// TIA Portal project "FactoryIO_Template_S7-1500_V14" (V14)

(* hardware
DEVICE "S71500/ET200MP-Station_1"  S7-1500 station
   slot 0: "Profilschiene_0"  6ES7 590-1***0-0AA0
   slot 1: "PLC_1"  CPU 1511-1 PN  6ES7 511-1AK00-0AB0  V1.8
   slot 2: "AI 8xU/I/RTD/TC ST_1"  AI 8xU/I/RTD/TC ST  6ES7 531-7KF00-0AB0  V2.0
   slot 3: "AI 8xU/I/RTD/TC ST_2"  AI 8xU/I/RTD/TC ST  6ES7 531-7KF00-0AB0  V2.0
   slot 4: "AI 8xU/I/RTD/TC ST_3"  AI 8xU/I/RTD/TC ST  6ES7 531-7KF00-0AB0  V2.0
   slot 5: "AI 8xU/I/RTD/TC ST_4"  AI 8xU/I/RTD/TC ST  6ES7 531-7KF00-0AB0  V2.0
   slot 6: "DI 16x24VDC BA_1"  DI 16x24VDC BA  6ES7 521-1BH10-0AA0  V1.0
*)

// ===== PLC "PLC_1"  CPU 1511-1 PN =====

VAR_GLOBAL   // PLC tag table "Standard-Variablentabelle"
   "start button" AT %I0.0 : Bool;
   "konveyöl 1" AT %Q0.0 : Bool;
   "start ışık" AT %Q0.1 : Bool;
   "Stop button" AT %I0.1 : Bool;
   "stop ışık" AT %Q0.2 : Bool;
   "mavi metaryel sensor" AT %I0.2 : Bool;
   "konveyör mavi yol" AT %Q0.3 : Bool;
   "mavi kemer" AT %Q0.4 : Bool;
   "mavi kol" AT %Q0.5 : Bool;
   "mavi bekleme" AT %Q0.6 : Bool;
   "mavi bekleme sensör baş" AT %I0.3 : Bool;
   "mavie bekleme sensör son" AT %I0.4 : Bool;
   "mavi x hareket" AT %Q0.7 : Bool;
   "mavi hareket z" AT %Q1.0 : Bool;
   "mavi tutucu(1)" AT %Q1.1 : Bool;
   "restart" AT %I0.5 : Bool;
   "depo mavi" AT %Q1.2 : Bool;
   "depo mavi sensor" AT %I0.6 : Bool;
   "mavi depo lamba" AT %Q1.3 : Bool;
   "mavi restart" AT %I0.7 : Bool;
   "konveyör 2" AT %Q1.4 : Bool;
   "konveyör yeşil yol" AT %Q1.5 : Bool;
   "yeşil metaryel sensör" AT %I1.0 : Bool;
   "yeşil kol" AT %Q1.6 : Bool;
   "yeşil kemer" AT %Q1.7 : Bool;
   "yeşil bekleme sensör baş" AT %I1.1 : Bool;
   "yeşil bekleme sensör son" AT %I1.2 : Bool;
   "yeşil bekleme" AT %Q2.0 : Bool;
   "depo mavi sensör" AT %I1.3 : Bool;
   "yeşil x hareket" AT %Q2.1 : Bool;
   "yeşil hareket z" AT %Q2.2 : Bool;
   "yeşil tutucu(1)" AT %Q2.3 : Bool;
   "depo yeşil sensor" AT %I1.4 : Bool;
   "yeşil restart" AT %I1.5 : Bool;
   "depo yeşil" AT %Q2.4 : Bool;
   "depo yeşil lamba" AT %Q2.5 : Bool;
   "Tag_1" AT %M110.0 : Bool;
   "Tag_2" AT %M120.0 : Bool;
   "konveyör metal yol" AT %Q2.6 : Bool;
   "metal metaryel sensör" AT %I1.6 : Bool;
   "metal kol" AT %Q2.7 : Bool;
   "metal kemer" AT %Q3.0 : Bool;
   "metal bekleme baş" AT %I1.7 : Bool;
   "metal bekleme son" AT %I2.0 : Bool;
   "metal bekleme" AT %Q3.1 : Bool;
   "depo metal sensör" AT %I2.1 : Bool;
   "depo metal" AT %Q3.5 : Bool;
   "depo metal lamba" AT %Q3.6 : Bool;
   "Tag_3" AT %M130.0 : Bool;
   "metal restart" AT %I2.2 : Bool;
   "Tag_4" AT %MD140 : Real;
   "Tag_5" AT %QW30 : Word;
   "metal y" AT %QD30 : Real;
   "Tag_7" AT %MD150 : Real;
   "metal z" AT %QD34 : Real;
   "metal tutma" AT %Q3.2 : Bool;
   "Tag_9" AT %MD160 : Real;
   "metal x" AT %QD38 : Real;
END_VAR

// folder: System blocks/Program resources

DATA_BLOCK "mavi"   // DB1
{ S7_Optimized_Access := 'TRUE' }
AUTHOR : Simatic
FAMILY : IEC
NAME : IEC_TMR
VERSION : 1.0
// stored: InstanceOfName IEC_TIMER
"IEC_TIMER"
BEGIN
END_DATA_BLOCK

DATA_BLOCK "mavi depolama"   // DB2
{ S7_Optimized_Access := 'TRUE' }
AUTHOR : Simatic
FAMILY : IEC
NAME : IEC_TMR
VERSION : 1.0
// stored: InstanceOfName IEC_TIMER
"IEC_TIMER"
BEGIN
END_DATA_BLOCK

DATA_BLOCK "mavi tutucu"   // DB3
{ S7_Optimized_Access := 'TRUE' }
AUTHOR : Simatic
FAMILY : IEC
NAME : IEC_TMR
VERSION : 1.0
// stored: InstanceOfName IEC_TIMER
"IEC_TIMER"
BEGIN
END_DATA_BLOCK

DATA_BLOCK "mavi 2"   // DB4
{ S7_Optimized_Access := 'TRUE' }
AUTHOR : Simatic
FAMILY : IEC
NAME : IEC_TMR
VERSION : 1.0
// stored: InstanceOfName IEC_TIMER
"IEC_TIMER"
BEGIN
END_DATA_BLOCK

DATA_BLOCK "mavi 3"   // DB5
{ S7_Optimized_Access := 'TRUE' }
AUTHOR : Simatic
FAMILY : IEC
NAME : IEC_TMR
VERSION : 1.0
// stored: InstanceOfName IEC_TIMER
"IEC_TIMER"
BEGIN
END_DATA_BLOCK

DATA_BLOCK "mavi 4"   // DB6
{ S7_Optimized_Access := 'TRUE' }
AUTHOR : Simatic
FAMILY : IEC
NAME : IEC_TMR
VERSION : 1.0
// stored: InstanceOfName IEC_TIMER
"IEC_TIMER"
BEGIN
END_DATA_BLOCK

DATA_BLOCK "mavi bekleme son sayıcı"   // DB7
{ S7_Optimized_Access := 'TRUE' }
AUTHOR : Simatic
FAMILY : IEC
NAME : CNTR
VERSION : 1.0
// stored: InstanceOfName IEC_COUNTER
"IEC_COUNTER"
BEGIN
END_DATA_BLOCK

DATA_BLOCK "yeşil"   // DB8
{ S7_Optimized_Access := 'TRUE' }
AUTHOR : Simatic
FAMILY : IEC
NAME : IEC_TMR
VERSION : 1.0
// stored: InstanceOfName IEC_TIMER
"IEC_TIMER"
BEGIN
END_DATA_BLOCK

DATA_BLOCK "yeşil depolama"   // DB9
{ S7_Optimized_Access := 'TRUE' }
AUTHOR : Simatic
FAMILY : IEC
NAME : IEC_TMR
VERSION : 1.0
// stored: InstanceOfName IEC_TIMER
"IEC_TIMER"
BEGIN
END_DATA_BLOCK

DATA_BLOCK "yeşil tutucu"   // DB10
{ S7_Optimized_Access := 'TRUE' }
AUTHOR : Simatic
FAMILY : IEC
NAME : IEC_TMR
VERSION : 1.0
// stored: InstanceOfName IEC_TIMER
"IEC_TIMER"
BEGIN
END_DATA_BLOCK

DATA_BLOCK "yeşil 2"   // DB11
{ S7_Optimized_Access := 'TRUE' }
AUTHOR : Simatic
FAMILY : IEC
NAME : IEC_TMR
VERSION : 1.0
// stored: InstanceOfName IEC_TIMER
"IEC_TIMER"
BEGIN
END_DATA_BLOCK

DATA_BLOCK "yeşil 3"   // DB12
{ S7_Optimized_Access := 'TRUE' }
AUTHOR : Simatic
FAMILY : IEC
NAME : IEC_TMR
VERSION : 1.0
// stored: InstanceOfName IEC_TIMER
"IEC_TIMER"
BEGIN
END_DATA_BLOCK

DATA_BLOCK "yeşil 4"   // DB13
{ S7_Optimized_Access := 'TRUE' }
AUTHOR : Simatic
FAMILY : IEC
NAME : IEC_TMR
VERSION : 1.0
// stored: InstanceOfName IEC_TIMER
"IEC_TIMER"
BEGIN
END_DATA_BLOCK

DATA_BLOCK "yeşil bekleme son sayıcı"   // DB14
{ S7_Optimized_Access := 'TRUE' }
AUTHOR : Simatic
FAMILY : IEC
NAME : CNTR
VERSION : 1.0
// stored: InstanceOfName IEC_COUNTER
"IEC_COUNTER"
BEGIN
END_DATA_BLOCK

DATA_BLOCK "mavi sayma"   // DB15
{ S7_Optimized_Access := 'TRUE' }
AUTHOR : Simatic
FAMILY : IEC
NAME : IEC_TMR
VERSION : 1.0
// stored: InstanceOfName IEC_TIMER
"IEC_TIMER"
BEGIN
END_DATA_BLOCK

DATA_BLOCK "yeşil sayma"   // DB16
{ S7_Optimized_Access := 'TRUE' }
AUTHOR : Simatic
FAMILY : IEC
NAME : IEC_TMR
VERSION : 1.0
// stored: InstanceOfName IEC_TIMER
"IEC_TIMER"
BEGIN
END_DATA_BLOCK

DATA_BLOCK "metal"   // DB17
{ S7_Optimized_Access := 'TRUE' }
AUTHOR : Simatic
FAMILY : IEC
NAME : IEC_TMR
VERSION : 1.0
// stored: InstanceOfName IEC_TIMER
"IEC_TIMER"
BEGIN
END_DATA_BLOCK

DATA_BLOCK "metal 1"   // DB18
{ S7_Optimized_Access := 'TRUE' }
AUTHOR : Simatic
FAMILY : IEC
NAME : IEC_TMR
VERSION : 1.0
// stored: InstanceOfName IEC_TIMER
"IEC_TIMER"
BEGIN
END_DATA_BLOCK

DATA_BLOCK "metal 2"   // DB19
{ S7_Optimized_Access := 'TRUE' }
AUTHOR : Simatic
FAMILY : IEC
NAME : IEC_TMR
VERSION : 1.0
// stored: InstanceOfName IEC_TIMER
"IEC_TIMER"
BEGIN
END_DATA_BLOCK

DATA_BLOCK "metal 3"   // DB20
{ S7_Optimized_Access := 'TRUE' }
AUTHOR : Simatic
FAMILY : IEC
NAME : IEC_TMR
VERSION : 1.0
// stored: InstanceOfName IEC_TIMER
"IEC_TIMER"
BEGIN
END_DATA_BLOCK

DATA_BLOCK "metal 4"   // DB21
{ S7_Optimized_Access := 'TRUE' }
AUTHOR : Simatic
FAMILY : IEC
NAME : IEC_TMR
VERSION : 1.0
// stored: InstanceOfName IEC_TIMER
"IEC_TIMER"
BEGIN
END_DATA_BLOCK

DATA_BLOCK "metal 5"   // DB22
{ S7_Optimized_Access := 'TRUE' }
AUTHOR : Simatic
FAMILY : IEC
NAME : IEC_TMR
VERSION : 1.0
// stored: InstanceOfName IEC_TIMER
"IEC_TIMER"
BEGIN
END_DATA_BLOCK

DATA_BLOCK "metal bekleme son sayıcı"   // DB23
{ S7_Optimized_Access := 'TRUE' }
AUTHOR : Simatic
FAMILY : IEC
NAME : CNTR
VERSION : 1.0
// stored: InstanceOfName IEC_COUNTER
"IEC_COUNTER"
BEGIN
END_DATA_BLOCK

DATA_BLOCK "metal sayma"   // DB24
{ S7_Optimized_Access := 'TRUE' }
AUTHOR : Simatic
FAMILY : IEC
NAME : IEC_TMR
VERSION : 1.0
// stored: InstanceOfName IEC_TIMER
"IEC_TIMER"
BEGIN
END_DATA_BLOCK

// folder: (top level)

FUNCTION "MHJ-PLC-Lab-Function-S71500" : Void   // FC9000, SCL
{ S7_Optimized_Access := 'TRUE' }
VERSION : 0.1
   VAR_TEMP
      Value : Byte;
      ForCounter : Int;
   END_VAR
   VAR CONSTANT
      Value_01_DW : DWord := 16#1223_5486;
      Value_02_DW : DWord := 16#A6C9_D1F5;
   END_VAR
BEGIN

   #Value:=PEEK(area := 16#82,
        dbNumber := 0,
        byteOffset := 511);
   #Value := #Value + 1;

   POKE(area := 16#82,
        dbNumber := 0,
        byteOffset := 511,
        value := #Value);

   POKE(area := 16#82,
        dbNumber := 0,
        byteOffset := 1016,
        value := #Value_01_DW);
   POKE(area := 16#82,
        dbNumber := 0,
        byteOffset := 1020,
        value := #Value_02_DW);

   FOR #ForCounter := 0 TO 63 DO
       #Value:=PEEK(area := 16#1,
            dbNumber := 0,
            byteOffset := #ForCounter);
       POKE(area := 16#81,
            dbNumber := 0,
            byteOffset := #ForCounter,
            value := #Value);
   END_FOR;
   #Value := PEEK(area := 16#1,
                  dbNumber := 0,
                  byteOffset := 512);
   POKE(area := 16#82,
        dbNumber := 0,
        byteOffset := 512,
        value := #Value);
END_FUNCTION

ORGANIZATION_BLOCK "Main"   // OB1, LAD, ProgramCycle
TITLE = "Main Program Sweep (Cycle)"
{ S7_Optimized_Access := 'TRUE' }
VERSION : 0.1
   VAR_INPUT
      Initial_Call : Bool;   // Initial call of this OB
      Remanence : Bool;   // =True, if remanent data are available
   END_VAR
   VAR_TEMP   // added for the SCL form of the ladder/FBD networks
      _w1 : Bool;
      _w2 : Bool;
   END_VAR
BEGIN

REGION Network 1
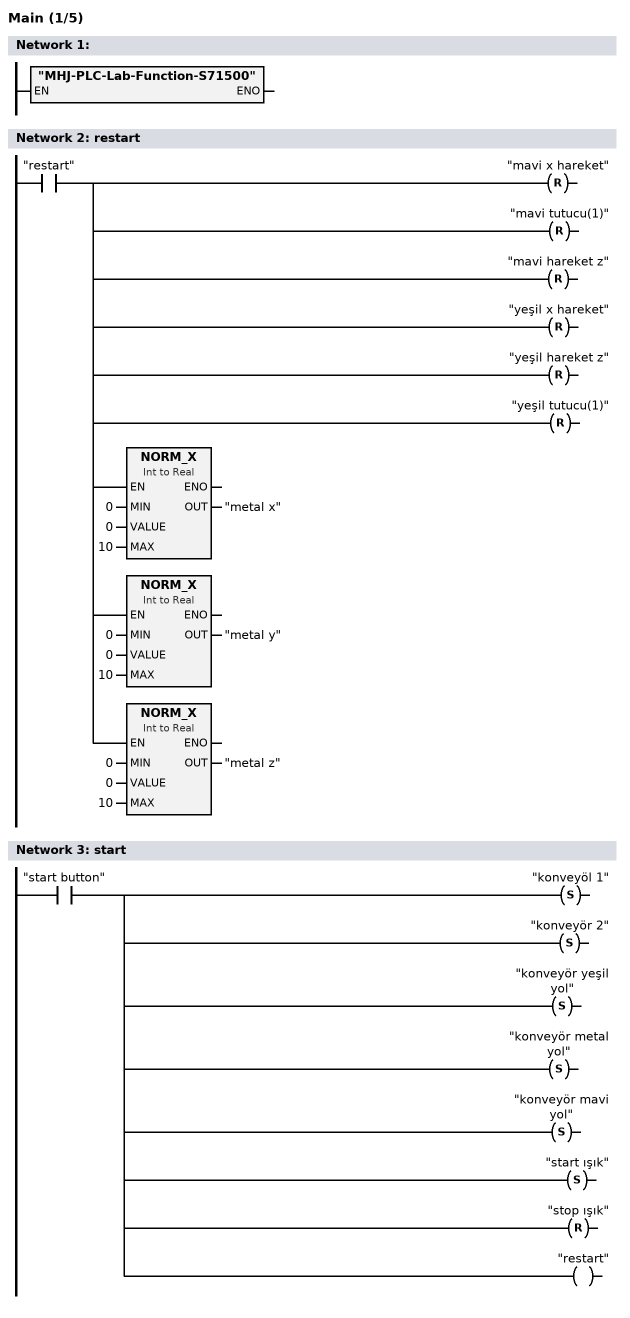
   RUNG wire#powerrail
      "MHJ-PLC-Lab-Function-S71500"()
   END_RUNG
   // the same network as SCL:
   "MHJ-PLC-Lab-Function-S71500"();
END_REGION

REGION Network 2: restart
   RUNG wire#powerrail
      Contact( "restart" )
      wire#w1
      R_Coil( "mavi x hareket" )
   END_RUNG
   RUNG wire#w1
      R_Coil( "mavi tutucu(1)" )
   END_RUNG
   RUNG wire#w1
      R_Coil( "mavi hareket z" )
   END_RUNG
   RUNG wire#w1
      R_Coil( "yeşil x hareket" )
   END_RUNG
   RUNG wire#w1
      R_Coil( "yeşil hareket z" )
   END_RUNG
   RUNG wire#w1
      R_Coil( "yeşil tutucu(1)" )
   END_RUNG
   RUNG wire#w1
      { S7_Templates := "[SrcType := Int, DestType := Real]" } Normalize(min := 0, value := 0, max := 10, out => "metal x")
   END_RUNG
   RUNG wire#w1
      { S7_Templates := "[SrcType := Int, DestType := Real]" } Normalize(min := 0, value := 0, max := 10, out => "metal y")
   END_RUNG
   RUNG wire#w1
      { S7_Templates := "[SrcType := Int, DestType := Real]" } Normalize(min := 0, value := 0, max := 10, out => "metal z")
   END_RUNG
   // the same network as SCL:
   IF "restart" THEN
       "mavi x hareket" := FALSE;
       "mavi tutucu(1)" := FALSE;
       "mavi hareket z" := FALSE;
       "yeşil x hareket" := FALSE;
       "yeşil hareket z" := FALSE;
       "yeşil tutucu(1)" := FALSE;
       "metal x" := NORM_X(MIN := 0, VALUE := 0, MAX := 10);
       "metal y" := NORM_X(MIN := 0, VALUE := 0, MAX := 10);
       "metal z" := NORM_X(MIN := 0, VALUE := 0, MAX := 10);
   END_IF;
END_REGION

REGION Network 3: start
   RUNG wire#powerrail
      Contact( "start button" )
      wire#w1
      S_Coil( "konveyöl 1" )
   END_RUNG
   RUNG wire#w1
      S_Coil( "konveyör 2" )
   END_RUNG
   RUNG wire#w1
      S_Coil( "konveyör yeşil yol" )
   END_RUNG
   RUNG wire#w1
      S_Coil( "konveyör metal yol" )
   END_RUNG
   RUNG wire#w1
      S_Coil( "konveyör mavi yol" )
   END_RUNG
   RUNG wire#w1
      S_Coil( "start ışık" )
   END_RUNG
   RUNG wire#w1
      R_Coil( "stop ışık" )
   END_RUNG
   RUNG wire#w1
      Coil( "restart" )
   END_RUNG
   // the same network as SCL:
   IF "start button" THEN
       "konveyöl 1" := TRUE;
       "konveyör 2" := TRUE;
       "konveyör yeşil yol" := TRUE;
       "konveyör metal yol" := TRUE;
       "konveyör mavi yol" := TRUE;
       "start ışık" := TRUE;
       "stop ışık" := FALSE;
   END_IF;
   "restart" := "start button";
END_REGION

REGION Network 4: stop
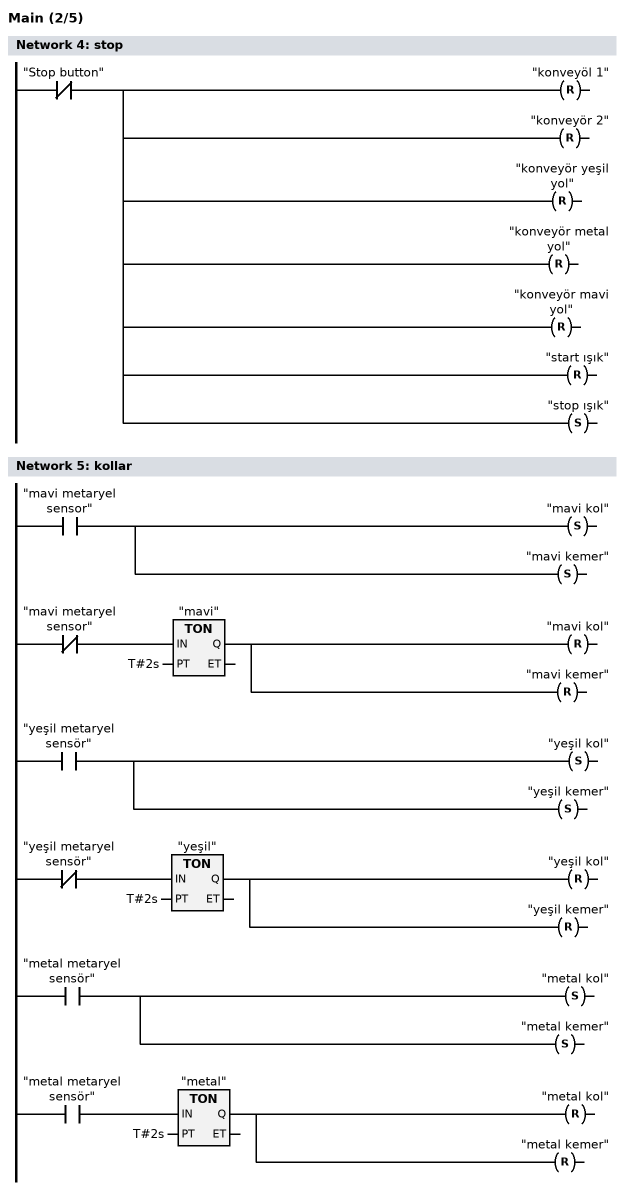
   RUNG wire#powerrail
      I_Contact( "Stop button" )
      wire#w1
      R_Coil( "konveyöl 1" )
   END_RUNG
   RUNG wire#w1
      R_Coil( "konveyör 2" )
   END_RUNG
   RUNG wire#w1
      R_Coil( "konveyör yeşil yol" )
   END_RUNG
   RUNG wire#w1
      R_Coil( "konveyör metal yol" )
   END_RUNG
   RUNG wire#w1
      R_Coil( "konveyör mavi yol" )
   END_RUNG
   RUNG wire#w1
      R_Coil( "start ışık" )
   END_RUNG
   RUNG wire#w1
      S_Coil( "stop ışık" )
   END_RUNG
   // the same network as SCL:
   IF NOT "Stop button" THEN
       "konveyöl 1" := FALSE;
       "konveyör 2" := FALSE;
       "konveyör yeşil yol" := FALSE;
       "konveyör metal yol" := FALSE;
       "konveyör mavi yol" := FALSE;
       "start ışık" := FALSE;
       "stop ışık" := TRUE;
   END_IF;
END_REGION

REGION Network 5: kollar
   IF "mavi metaryel sensor" THEN
       "mavi kol" := TRUE;
       "mavi kemer" := TRUE;
   END_IF;
   "mavi".TON(IN := NOT "mavi metaryel sensor", PT := T#2s);
   IF "mavi".Q THEN
       "mavi kol" := FALSE;
       "mavi kemer" := FALSE;
   END_IF;
   IF "yeşil metaryel sensör" THEN
       "yeşil kol" := TRUE;
       "yeşil kemer" := TRUE;
   END_IF;
   "yeşil".TON(IN := NOT "yeşil metaryel sensör", PT := T#2s);
   IF "yeşil".Q THEN
       "yeşil kol" := FALSE;
       "yeşil kemer" := FALSE;
   END_IF;
   IF "metal metaryel sensör" THEN
       "metal kol" := TRUE;
       "metal kemer" := TRUE;
   END_IF;
   "metal".TON(IN := "metal metaryel sensör", PT := T#2s);
   IF "metal".Q THEN
       "metal kol" := FALSE;
       "metal kemer" := FALSE;
   END_IF;
END_REGION

REGION Network 6: bekleme
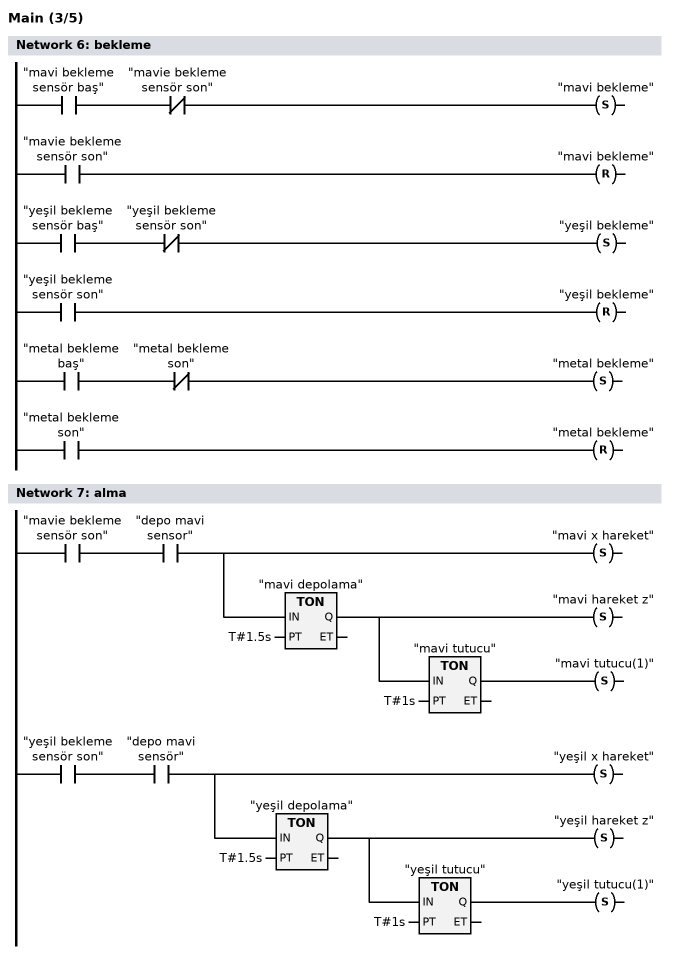
   RUNG wire#powerrail
      Contact( "mavi bekleme sensör baş" )
      I_Contact( "mavie bekleme sensör son" )
      S_Coil( "mavi bekleme" )
   END_RUNG
   RUNG wire#powerrail
      Contact( "mavie bekleme sensör son" )
      R_Coil( "mavi bekleme" )
   END_RUNG
   RUNG wire#powerrail
      Contact( "yeşil bekleme sensör baş" )
      I_Contact( "yeşil bekleme sensör son" )
      S_Coil( "yeşil bekleme" )
   END_RUNG
   RUNG wire#powerrail
      Contact( "yeşil bekleme sensör son" )
      R_Coil( "yeşil bekleme" )
   END_RUNG
   RUNG wire#powerrail
      Contact( "metal bekleme baş" )
      I_Contact( "metal bekleme son" )
      S_Coil( "metal bekleme" )
   END_RUNG
   RUNG wire#powerrail
      Contact( "metal bekleme son" )
      R_Coil( "metal bekleme" )
   END_RUNG
   // the same network as SCL:
   IF "mavi bekleme sensör baş" AND NOT "mavie bekleme sensör son" THEN "mavi bekleme" := TRUE; END_IF;
   IF "mavie bekleme sensör son" THEN "mavi bekleme" := FALSE; END_IF;
   IF "yeşil bekleme sensör baş" AND NOT "yeşil bekleme sensör son" THEN "yeşil bekleme" := TRUE; END_IF;
   IF "yeşil bekleme sensör son" THEN "yeşil bekleme" := FALSE; END_IF;
   IF "metal bekleme baş" AND NOT "metal bekleme son" THEN "metal bekleme" := TRUE; END_IF;
   IF "metal bekleme son" THEN "metal bekleme" := FALSE; END_IF;
END_REGION

REGION Network 7: alma
   #_w1 := "mavie bekleme sensör son" AND "depo mavi sensor";
   IF #_w1 THEN "mavi x hareket" := TRUE; END_IF;
   "mavi depolama".TON(IN := #_w1, PT := T#1.5s);
   IF "mavi depolama".Q THEN "mavi hareket z" := TRUE; END_IF;
   "mavi tutucu".TON(IN := "mavi depolama".Q, PT := T#1s);
   IF "mavi tutucu".Q THEN "mavi tutucu(1)" := TRUE; END_IF;
   #_w2 := "yeşil bekleme sensör son" AND "depo mavi sensör";
   IF #_w2 THEN "yeşil x hareket" := TRUE; END_IF;
   "yeşil depolama".TON(IN := #_w2, PT := T#1.5s);
   IF "yeşil depolama".Q THEN "yeşil hareket z" := TRUE; END_IF;
   "yeşil tutucu".TON(IN := "yeşil depolama".Q, PT := T#1s);
   IF "yeşil tutucu".Q THEN "yeşil tutucu(1)" := TRUE; END_IF;
END_REGION

REGION Network 8: birakma
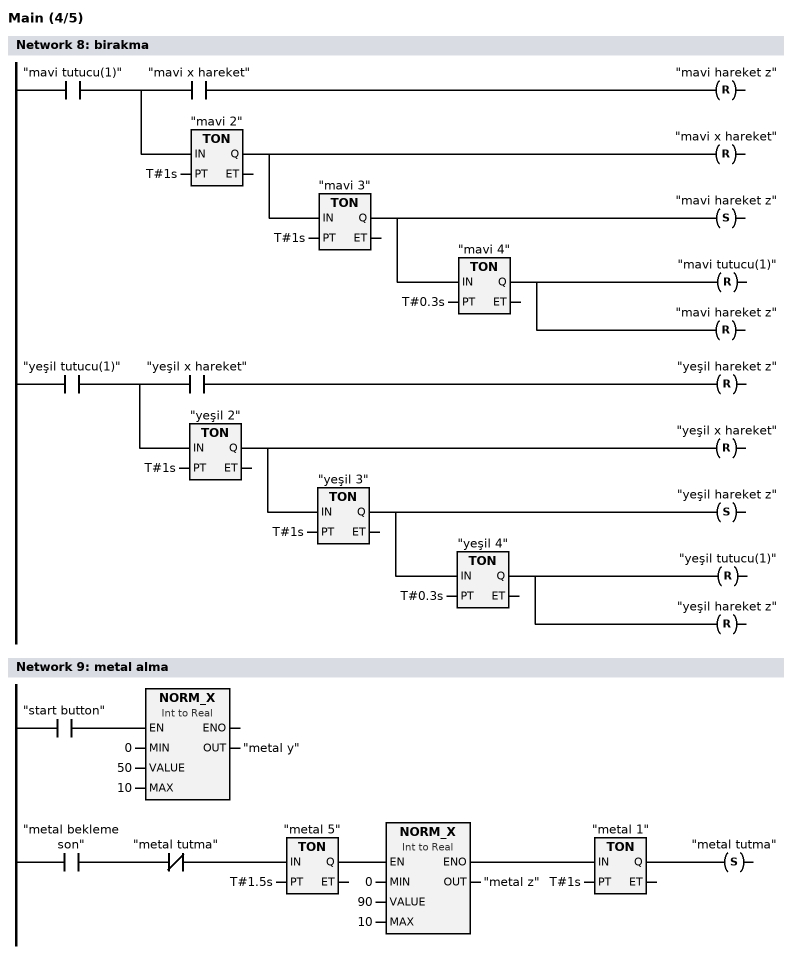
   IF "mavi tutucu(1)" AND "mavi x hareket" THEN "mavi hareket z" := FALSE; END_IF;
   "mavi 2".TON(IN := "mavi tutucu(1)", PT := T#1s);
   IF "mavi 2".Q THEN "mavi x hareket" := FALSE; END_IF;
   "mavi 3".TON(IN := "mavi 2".Q, PT := T#1s);
   IF "mavi 3".Q THEN "mavi hareket z" := TRUE; END_IF;
   "mavi 4".TON(IN := "mavi 3".Q, PT := T#0.3s);
   IF "mavi 4".Q THEN
       "mavi tutucu(1)" := FALSE;
       "mavi hareket z" := FALSE;
   END_IF;
   IF "yeşil tutucu(1)" AND "yeşil x hareket" THEN "yeşil hareket z" := FALSE; END_IF;
   "yeşil 2".TON(IN := "yeşil tutucu(1)", PT := T#1s);
   IF "yeşil 2".Q THEN "yeşil x hareket" := FALSE; END_IF;
   "yeşil 3".TON(IN := "yeşil 2".Q, PT := T#1s);
   IF "yeşil 3".Q THEN "yeşil hareket z" := TRUE; END_IF;
   "yeşil 4".TON(IN := "yeşil 3".Q, PT := T#0.3s);
   IF "yeşil 4".Q THEN
       "yeşil tutucu(1)" := FALSE;
       "yeşil hareket z" := FALSE;
   END_IF;
END_REGION

REGION Network 9: metal alma
   IF "start button" THEN "metal y" := NORM_X(MIN := 0, VALUE := 50, MAX := 10); END_IF;
   "metal 5".TON(IN := "metal bekleme son" AND NOT "metal tutma", PT := T#1.5s);
   IF "metal 5".Q THEN "metal z" := NORM_X(MIN := 0, VALUE := 90, MAX := 10); END_IF;
   "metal 1".TON(IN := "metal 5".Q, PT := T#1s);
   IF "metal 1".Q THEN "metal tutma" := TRUE; END_IF;
END_REGION

REGION Network 10: metal birakma
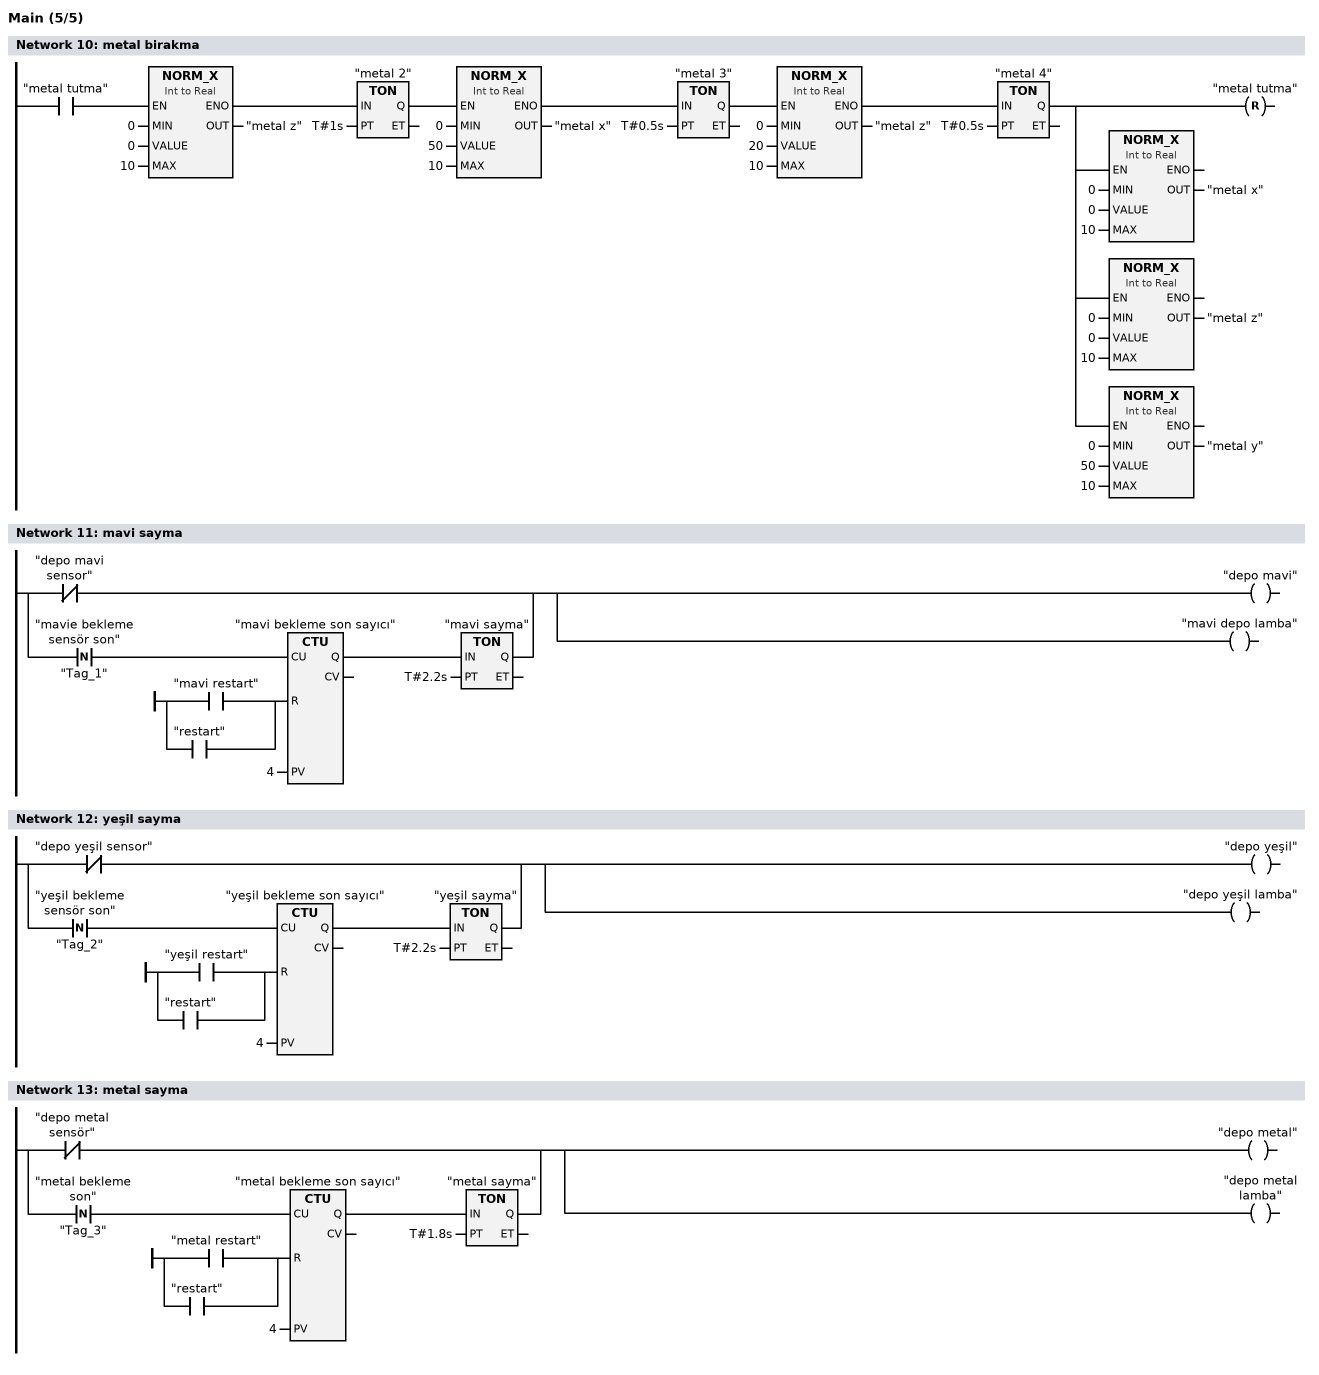
   IF "metal tutma" THEN "metal z" := NORM_X(MIN := 0, VALUE := 0, MAX := 10); END_IF;
   "metal 2".TON(IN := "metal tutma", PT := T#1s);
   IF "metal 2".Q THEN "metal x" := NORM_X(MIN := 0, VALUE := 50, MAX := 10); END_IF;
   "metal 3".TON(IN := "metal 2".Q, PT := T#0.5s);
   IF "metal 3".Q THEN "metal z" := NORM_X(MIN := 0, VALUE := 20, MAX := 10); END_IF;
   "metal 4".TON(IN := "metal 3".Q, PT := T#0.5s);
   IF "metal 4".Q THEN
       "metal tutma" := FALSE;
       "metal x" := NORM_X(MIN := 0, VALUE := 0, MAX := 10);
       "metal z" := NORM_X(MIN := 0, VALUE := 0, MAX := 10);
       "metal y" := NORM_X(MIN := 0, VALUE := 50, MAX := 10);
   END_IF;
END_REGION

REGION Network 11: mavi sayma
   #_w1 := NOT "mavie bekleme sensör son" AND "Tag_1";   // falling edge of "mavie bekleme sensör son"
   "Tag_1" := "mavie bekleme sensör son";
   "mavi bekleme son sayıcı".CTU(CU := #_w1, R := "mavi restart" OR "restart", PV := 4);
   "mavi sayma".TON(IN := "mavi bekleme son sayıcı".Q, PT := T#2.2s);
   "depo mavi" := NOT "depo mavi sensor" OR "mavi sayma".Q;
   "mavi depo lamba" := "depo mavi";
END_REGION

REGION Network 12: yeşil sayma
   #_w1 := NOT "yeşil bekleme sensör son" AND "Tag_2";   // falling edge of "yeşil bekleme sensör son"
   "Tag_2" := "yeşil bekleme sensör son";
   "yeşil bekleme son sayıcı".CTU(CU := #_w1, R := "yeşil restart" OR "restart", PV := 4);
   "yeşil sayma".TON(IN := "yeşil bekleme son sayıcı".Q, PT := T#2.2s);
   "depo yeşil" := NOT "depo yeşil sensor" OR "yeşil sayma".Q;
   "depo yeşil lamba" := "depo yeşil";
END_REGION

REGION Network 13: metal sayma
   #_w1 := NOT "metal bekleme son" AND "Tag_3";   // falling edge of "metal bekleme son"
   "Tag_3" := "metal bekleme son";
   "metal bekleme son sayıcı".CTU(CU := #_w1, R := "metal restart" OR "restart", PV := 4);
   "metal sayma".TON(IN := "metal bekleme son sayıcı".Q, PT := T#1.8s);
   "depo metal" := NOT "depo metal sensör" OR "metal sayma".Q;
   "depo metal lamba" := "depo metal";
END_REGION
END_ORGANIZATION_BLOCK